(*********************************** G.D S.p.A. - Technical Department ***********************************
============= PROGRAM INFO ============
FOLDER:             TBD
MACHINES INVOLVED:  TBD 

============= DESCRIPTION =============
csp machine declaration

============= REVISIONS ===============
Date		Version	 	Author      	Description             
----------	-------		------------  	--------------------------------------------
2019/04/05 	0000.00	 	M.Grasso		Creation of the PRG

**********************************************************************************************************)
(*$R process_ref := prc; $*)
PROGRAM csp_case_fc_ls_upper
VAR
	
	prc:											process;
	prc_path:										STRING;
	
END_VAR

_read_var_input();

_object_manager();

IF NOT objects_running()
THEN
	RETURN;	
END_IF

_read_process_image();

_mode_manager();

_set_runtime_properties();

(********************************* BODY *********************************)
(************************************************************************)

_handle_messages();

_write_output();

ACTION _handle_messages:
;
END_ACTION

ACTION _handle_process_test:
;
END_ACTION

ACTION _mode_manager:
IF process_mode_req_is_pending(prc)
THEN
    process_apply_mode_req_first_step(prc);
    CASE process_get_mode(prc) OF
        MODE_TO_ABSENT:
			;
        MODE_TO_INACTIVE:
			;
        MODE_TO_TEST:
			;
        MODE_TO_OPERATIONAL:
			;
    END_CASE
    process_apply_mode_req_second_step(prc);
END_IF
END_ACTION

ACTION _object_manager:
IF objects_initialization()
THEN
	sub_process_init(
		object_name					:= 'csp_case_fc_ls_upper.prc', 
		process						:= csp_case_flapControl_ls.prc, 
		CONVERSION_this				:= prc);
		
	prc_path 						:= process_get_path(prc);
END_IF

IF objects_running()
THEN
	process_cycle(prc);
END_IF
END_ACTION

ACTION _read_process_image:
;
END_ACTION

ACTION _read_var_input:
;
END_ACTION

ACTION _set_runtime_properties:
;
END_ACTION

ACTION _write_output:
;
END_ACTION

END_PROGRAM

(* stored: Version 1.1.0.1, ProductVersion 3.1.4022.12
   POU csp_case_fc_ls_upper: Id {603f3961-01f1-4b8e-91d3-f76591b087d3}, SpecialFunc None
   Action _handle_messages: Id {bab5a346-1bd1-429f-916e-5a9e81144aec}
   Action _handle_process_test: Id {6a65092a-4764-4754-94c7-a77d5f37cd8e}
   Action _mode_manager: Id {36a71676-fce0-4c19-b52a-f93119c43f2d}
   Action _object_manager: Id {4256983d-cc36-4c4e-b322-c45f00813b3e}
   Action _read_process_image: Id {987f1a28-e8ca-4e14-996f-ca456be512b4}
   Action _read_var_input: Id {f47fe7aa-8e93-4122-aee1-ae56fe04e72a}
   Action _set_runtime_properties: Id {8771e7e7-bfc7-4738-adc1-47f607633efd}
   Action _write_output: Id {2cead5b7-2d26-44a2-91d0-ef15b0c3f559} *)
